FUNCTION_BLOCK FieldSignals (* CAT Function Block Type *)
  (* Standard: 61499-2 *)
  (* Version 0.0, 3/5/2026, Schneider Electric, template *)
  PACKAGE SE.Nereda;
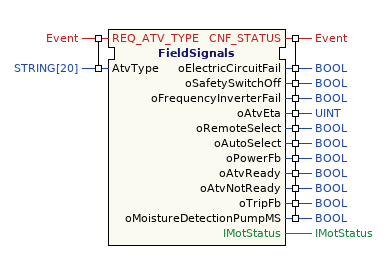
  EVENT_INPUT
    REQ_ATV_TYPE WITH AtvType;
  END_EVENT
  EVENT_OUTPUT
    CNF_STATUS WITH oElectricCircuitFail, oSafetySwitchOff, oFrequencyInverterFail, oAtvEta, oRemoteSelect, oAutoSelect, oPowerFb, oAtvReady, oAtvNotReady, oTripFb, oMoistureDetectionPumpMS;
  END_EVENT
  VAR_INPUT
    AtvType : STRING[20];
  END_VAR
  VAR_OUTPUT
    oElectricCircuitFail : BOOL; (* Current value(i) in the named variable array element *)
    oSafetySwitchOff : BOOL; (* Current value(i) in the named variable array element *)
    oFrequencyInverterFail : BOOL; (* Current value(i) in the named variable array element *)
    oAtvEta : UINT; (* Current value(i) in the named variable array element *)
    oRemoteSelect : BOOL; (* Current value(i) in the named variable array element *)
    oAutoSelect : BOOL; (* Current value(i) in the named variable array element *)
    oPowerFb : BOOL; (* Current value(i) in the named variable array element *)
    oAtvReady : BOOL; (* Current value(i) in the named variable array element *)
    oAtvNotReady : BOOL; (* Current value(i) in the named variable array element *)
    oTripFb : BOOL; (* Current value(i) in the named variable array element *)
    oMoistureDetectionPumpMS : BOOL;
  END_VAR
  PLUGS
    IMotStatus : IMotStatus;
  END_PLUGS
  (* 03 - FIELD INTERFACE IN *)
  (* 02 - FUNCTIONNAL OUTPUT INTERFACE *)
  (* 00 - INITIALIZATION *)
  (* 05 - LOGIC *)
  (* 04 - FIELD INTERFACE OUT *)
  (* 06 - HMI INTERFACE *)
  (* 01 - FUNCTIONNAL INPUT INTERFACE *)
  FBS
    INIT : plcStart(Prio := 24, Delay := T#0ms);
    ElectricCircuitFail : SYMLINKMULTIVARDST_1559B0FF8170C9BA0(QI := TRUE, NAME1 := '$${PATH}ElectricCircuitFail'); {SET_ATTRIBUTE(Configuration.GenericFBType.InterfaceParams, Runtime.System#I:=1;VALUE${I$}:BOOL)}
    SafetySwitchOff : SYMLINKMULTIVARDST_1559B0FF8170C9BA0(QI := TRUE, NAME1 := '$${PATH}SafetySwitchOff'); {SET_ATTRIBUTE(Configuration.GenericFBType.InterfaceParams, Runtime.System#I:=1;VALUE${I$}:BOOL)}
    FrequencyInverterFail : SYMLINKMULTIVARDST_1559B0FF8170C9BA0(QI := TRUE, NAME1 := '$${PATH}FrequencyInverterFail'); {SET_ATTRIBUTE(Configuration.GenericFBType.InterfaceParams, Runtime.System#I:=1;VALUE${I$}:BOOL)}
    ResetError_ATV3 : AtvResetError;
    ATV_ETA : SYMLINKMULTIVARDST_97F4072E4C409BE(QI := TRUE, NAME1 := '$${PATH}ATV_ETA'); {SET_ATTRIBUTE(Configuration.GenericFBType.InterfaceParams, Runtime.System#I:=1;VALUE${I$}:UINT)}
    ATV_Command : SYMLINKMULTIVARSRC_277E97BEC1451D2C(QI := TRUE, NAME1 := '$${PATH}ResetError_ATV', NAME2 := '$${PATH}CmdReady'); {SET_ATTRIBUTE(Configuration.GenericFBType.InterfaceParams, Runtime.System#I:=2;VALUE${I$}:BOOL,BOOL)}
    IThis : FieldSignals_HMI(QI := TRUE);
    RemoteSelect : SYMLINKMULTIVARDST_1559B0FF8170C9BA0(QI := TRUE, NAME1 := '$${PATH}RemoteSelect'); {SET_ATTRIBUTE(Configuration.GenericFBType.InterfaceParams, Runtime.System#I:=1;VALUE${I$}:BOOL)}
    AutoSelect : SYMLINKMULTIVARDST_1559B0FF8170C9BA0(QI := TRUE, NAME1 := '$${PATH}AutoSelect'); {SET_ATTRIBUTE(Configuration.GenericFBType.InterfaceParams, Runtime.System#I:=1;VALUE${I$}:BOOL)}
    PowerFb : SYMLINKMULTIVARDST_1559B0FF8170C9BA0(QI := TRUE, NAME1 := '$${PATH}PowerFb'); {SET_ATTRIBUTE(Configuration.GenericFBType.InterfaceParams, Runtime.System#I:=1;VALUE${I$}:BOOL)}
    AtvReady : SYMLINKMULTIVARDST_1559B0FF8170C9BA0(QI := TRUE, NAME1 := '$${PATH}AtvReady'); {SET_ATTRIBUTE(Configuration.GenericFBType.InterfaceParams, Runtime.System#I:=1;VALUE${I$}:BOOL)}
    EO_STATUS : E_MERGE_12;
    AtvNotReady : NOT_42C76073DCEB1A7A; {SET_ATTRIBUTE(Configuration.GenericFBType.InterfaceParams, Runtime.Standard#CNT:=1;OUT${CNT$}:BOOL)}
    RemoteAutoSelectMng : RemoteAutoMng;
    SelElectricCircuitFail : SELECT_81F91C08E00C8B28; {SET_ATTRIBUTE(Configuration.GenericFBType.InterfaceParams, Runtime.Standard#CNT:=2;SELECT:BOOL;IN${CNT$}:BOOL)}
    SelSafetySwitchOff : SELECT_81F91C08E00C8B28; {SET_ATTRIBUTE(Configuration.GenericFBType.InterfaceParams, Runtime.Standard#CNT:=2;SELECT:BOOL;IN${CNT$}:BOOL)}
    SelFrequencyInverterFail : SELECT_81F91C08E00C8B28; {SET_ATTRIBUTE(Configuration.GenericFBType.InterfaceParams, Runtime.Standard#CNT:=2;SELECT:BOOL;IN${CNT$}:BOOL)}
    SelATV_ETA : SELECT_32E1B08D4B0D0FE1; {SET_ATTRIBUTE(Configuration.GenericFBType.InterfaceParams, Runtime.Standard#CNT:=2;SELECT:BOOL;IN${CNT$}:UINT)}
    SelRemoteSelect : SELECT_81F91C08E00C8B28; {SET_ATTRIBUTE(Configuration.GenericFBType.InterfaceParams, Runtime.Standard#CNT:=2;SELECT:BOOL;IN${CNT$}:BOOL)}
    SelAutoSelect : SELECT_81F91C08E00C8B28; {SET_ATTRIBUTE(Configuration.GenericFBType.InterfaceParams, Runtime.Standard#CNT:=2;SELECT:BOOL;IN${CNT$}:BOOL)}
    SelPowerFb : SELECT_81F91C08E00C8B28; {SET_ATTRIBUTE(Configuration.GenericFBType.InterfaceParams, Runtime.Standard#CNT:=2;SELECT:BOOL;IN${CNT$}:BOOL)}
    SelAtvReady : SELECT_81F91C08E00C8B28; {SET_ATTRIBUTE(Configuration.GenericFBType.InterfaceParams, Runtime.Standard#CNT:=2;SELECT:BOOL;IN${CNT$}:BOOL)}
    NameGenerator : VALFORMAT_8708B18B173C5ABA(FORMAT := '%s', VALUE1 := '$${PATH:3,0}'); {SET_ATTRIBUTE(Configuration.GenericFBType.InterfaceParams, Runtime.Standard#I:=1;VALUE${I$}:STRING)}
    Frequency : SYMLINKMULTIVARDST_197068ABA215D7EBA(QI := TRUE, NAME1 := '$${PATH}MotorFrequecy'); {SET_ATTRIBUTE(Configuration.GenericFBType.InterfaceParams, Runtime.System#I:=1;VALUE${I$}:REAL)}
    PowerPercent_Sym : SYMLINKMULTIVARDST_197068ABA215D7EBA(QI := TRUE, NAME1 := '$${PATH}PowerPercent'); {SET_ATTRIBUTE(Configuration.GenericFBType.InterfaceParams, Runtime.System#I:=1;VALUE${I$}:REAL)}
    PowerCalculator : AtvPowerCalculator;
    TRIP : SYMLINKMULTIVARDST_1559B0FF8170C9BA0(QI := TRUE, NAME1 := '$${PATH}TRIP'); {SET_ATTRIBUTE(Configuration.GenericFBType.InterfaceParams, Runtime.System#I:=1;VALUE${I$}:BOOL)}
    SelTrip : SELECT_81F91C08E00C8B28; {SET_ATTRIBUTE(Configuration.GenericFBType.InterfaceParams, Runtime.Standard#CNT:=2;SELECT:BOOL;IN${CNT$}:BOOL)}
    MoistureDetectionPumpMS : SYMLINKMULTIVARDST_1559B0FF8170C9BA0(QI := TRUE, NAME1 := '$${PATH}MoistureDetectionPumpMS'); {SET_ATTRIBUTE(Configuration.GenericFBType.InterfaceParams, Runtime.System#I:=1;VALUE${I$}:BOOL)}
    SelMDPMS : SELECT_81F91C08E00C8B28; {SET_ATTRIBUTE(Configuration.GenericFBType.InterfaceParams, Runtime.Standard#CNT:=2;SELECT:BOOL;IN${CNT$}:BOOL)}
    NotElectricCircuitFail : NOT_42C76073DCEB1A7A; {SET_ATTRIBUTE(Configuration.GenericFBType.InterfaceParams, Runtime.Standard#CNT:=1;OUT${CNT$}:BOOL)}
    NOT1 : NOT_42C76073DCEB1A7A; {SET_ATTRIBUTE(Configuration.GenericFBType.InterfaceParams, Runtime.Standard#CNT:=1;OUT${CNT$}:BOOL)}
  END_FBS
  EVENT_CONNECTIONS
    ElectricCircuitFail.INITO TO SafetySwitchOff.INIT;
    SafetySwitchOff.INITO TO FrequencyInverterFail.INIT;
    FrequencyInverterFail.INITO TO ATV_ETA.INIT;
    ATV_ETA.INITO TO RemoteSelect.INIT;
    RemoteSelect.INITO TO AutoSelect.INIT;
    AutoSelect.INITO TO PowerFb.INIT;
    PowerFb.INITO TO AtvReady.INIT;
    SelAtvReady.CNF TO AtvNotReady.REQ;
    ElectricCircuitFail.CNF TO SelElectricCircuitFail.REQ;
    SafetySwitchOff.CNF TO SelSafetySwitchOff.REQ;
    FrequencyInverterFail.CNF TO SelFrequencyInverterFail.REQ;
    ATV_ETA.CNF TO SelATV_ETA.REQ;
    RemoteSelect.CNF TO SelRemoteSelect.REQ;
    AutoSelect.CNF TO SelAutoSelect.REQ;
    PowerFb.CNF TO SelPowerFb.REQ;
    AtvReady.CNF TO SelAtvReady.REQ;
    Frequency.INITO TO PowerPercent_Sym.INIT;
    AtvReady.INITO TO Frequency.INIT;
    PowerPercent_Sym.INITO TO TRIP.INIT;
    MoistureDetectionPumpMS.INITO TO ATV_Command.INIT;
    TRIP.CNF TO SelTrip.REQ;
    TRIP.INITO TO MoistureDetectionPumpMS.INIT;
    NOT1.CNF TO SelMDPMS.REQ;
    NotElectricCircuitFail.CNF TO IMotStatus.DA4A5AB166737E2B;
    SelSafetySwitchOff.CNF TO IMotStatus.SAF_SWT;
    SelFrequencyInverterFail.CNF TO IMotStatus.FREQ_FAIL;
    SelAtvReady.CNF TO IMotStatus.ATV_STE;
    SelRemoteSelect.CNF TO IMotStatus.REM_SEL;
    SelAutoSelect.CNF TO IMotStatus.AUTO_SEL;
    SelPowerFb.CNF TO IMotStatus.PWR_FB;
    SelTrip.CNF TO IMotStatus.8F309C1427B3D8B8;
    SelMDPMS.CNF TO IMotStatus.58CE25A170A20217;
    EO_STATUS.EO TO CNF_STATUS;
    NotElectricCircuitFail.CNF TO EO_STATUS.EI1;
    SelSafetySwitchOff.CNF TO EO_STATUS.EI2;
    SelFrequencyInverterFail.CNF TO EO_STATUS.EI3;
    SelATV_ETA.CNF TO EO_STATUS.EI4;
    RemoteAutoSelectMng.6BEF700BD5F898F8 TO EO_STATUS.EI5;
    SelPowerFb.CNF TO EO_STATUS.EI6;
    AtvNotReady.CNF TO EO_STATUS.523A3C57C3E4FA0F;
    SelTrip.CNF TO EO_STATUS.61E483B0D1B23F8E;
    SelMDPMS.CNF TO EO_STATUS.5434FC65F5B992C5;
    SelRemoteSelect.CNF TO RemoteAutoSelectMng.64070B2561E430BA;
    SelAutoSelect.CNF TO RemoteAutoSelectMng.64070B2561E430BA;
    PowerPercent_Sym.CNF TO PowerCalculator.REQ_POWER_PERC;
    REQ_ATV_TYPE TO PowerCalculator.REQ_ATV_TYPE;
    ATV_Command.INITO TO ResetError_ATV3.INIT;
    SelATV_ETA.CNF TO ResetError_ATV3.867B421BA90E2810;
    ResetError_ATV3.INITO TO INIT.ACK_FIRST;
    ResetError_ATV3.INITO TO NameGenerator.REQ;
    ResetError_ATV3.AD4F06CAB1B76C3D TO ATV_Command.REQ;
    ResetError_ATV3.3BE1C5BD951DD8A7 TO ATV_Command.REQ;
    SelElectricCircuitFail.CNF TO NotElectricCircuitFail.REQ;
    INIT.FIRST_INIT TO IThis.AD2A2FBE3D868A1D;
    INIT.REDO_INIT TO IThis.AD2A2FBE3D868A1D;
    PowerCalculator.CNF_POWER TO IThis.63337A003134C8E1;
    EO_STATUS.EO TO IThis.63337A003134C8E1;
    Frequency.CNF TO IThis.63337A003134C8E1;
    NameGenerator.CNF TO IThis.DAE3B0FAEAC06339;
    ResetError_ATV3.INITO TO IThis.213B97BD352AC6B9;
    IThis.047CDA631ACD0253 TO ElectricCircuitFail.INIT;
    IThis.9F0BB3507B1E4504 TO SelElectricCircuitFail.REQ;
    IThis.BE640CA1368FDF36 TO SelSafetySwitchOff.REQ;
    IThis.F7F6E0FF8EFA4B9E TO SelFrequencyInverterFail.REQ;
    IThis.1FE9183DAACAEFB7 TO SelATV_ETA.REQ;
    IThis.9B6E94ED39D931DA TO SelRemoteSelect.REQ;
    IThis.748EF2C5409B754A TO SelAutoSelect.REQ;
    IThis.DD989F023E0D2E7F TO SelPowerFb.REQ;
    IThis.C26243D045851266 TO SelAtvReady.REQ;
    IThis.DF011DEE9B6BC98A TO SelTrip.REQ;
    IThis.72F15890245A8D67 TO SelMDPMS.REQ;
    IThis.20926393FE3C273B TO SelElectricCircuitFail.REQ;
    IThis.20926393FE3C273B TO SelSafetySwitchOff.REQ;
    IThis.20926393FE3C273B TO SelFrequencyInverterFail.REQ;
    IThis.20926393FE3C273B TO SelATV_ETA.REQ;
    IThis.20926393FE3C273B TO SelRemoteSelect.REQ;
    IThis.20926393FE3C273B TO SelAutoSelect.REQ;
    IThis.20926393FE3C273B TO SelPowerFb.REQ;
    IThis.20926393FE3C273B TO SelAtvReady.REQ;
    IThis.20926393FE3C273B TO SelTrip.REQ;
    IThis.20926393FE3C273B TO SelMDPMS.REQ;
    AtvReady.CNF TO ResetError_ATV3.9E72FB83DA008EE6;
    MoistureDetectionPumpMS.CNF TO NOT1.REQ;
  END_CONNECTIONS
  DATA_CONNECTIONS
    NotElectricCircuitFail.OUT1 TO oElectricCircuitFail;
    SelSafetySwitchOff.OUT TO oSafetySwitchOff;
    SelFrequencyInverterFail.OUT TO oFrequencyInverterFail;
    SelATV_ETA.OUT TO oAtvEta;
    SelPowerFb.OUT TO oPowerFb;
    SelAtvReady.OUT TO oAtvReady;
    AtvNotReady.OUT1 TO oAtvNotReady;
    SelAtvReady.OUT TO AtvNotReady.IN1;
    ElectricCircuitFail.VALUE1 TO SelElectricCircuitFail.IN1;
    SafetySwitchOff.VALUE1 TO SelSafetySwitchOff.IN1;
    FrequencyInverterFail.VALUE1 TO SelFrequencyInverterFail.IN1;
    ATV_ETA.VALUE1 TO SelATV_ETA.IN1;
    RemoteSelect.VALUE1 TO SelRemoteSelect.IN1;
    AutoSelect.VALUE1 TO SelAutoSelect.IN1;
    PowerFb.VALUE1 TO SelPowerFb.IN1;
    AtvReady.VALUE1 TO SelAtvReady.IN1;
    TRIP.VALUE1 TO SelTrip.IN1;
    SelTrip.OUT TO oTripFb;
    NOT1.OUT1 TO SelMDPMS.IN1;
    SelMDPMS.OUT TO oMoistureDetectionPumpMS;
    NotElectricCircuitFail.OUT1 TO IMotStatus.9BFF267744CD9FD6;
    SelSafetySwitchOff.OUT TO IMotStatus.78CB3852B3811624;
    SelFrequencyInverterFail.OUT TO IMotStatus.D764D50DE95B92F7;
    SelAtvReady.OUT TO IMotStatus.469BA920D864796D;
    RemoteAutoSelectMng.35EEAE8FF93B7DBA TO IMotStatus.EF0659DE8FA343F8;
    RemoteAutoSelectMng.A72D9DB047E13611 TO IMotStatus.1313714BCA2AD84D;
    SelPowerFb.OUT TO IMotStatus.DFE83B4BA65B6F23;
    SelTrip.OUT TO IMotStatus.56D1AD5F30D2DBE7;
    SelMDPMS.OUT TO IMotStatus.6ADAD9BF6A0BA01D;
    RemoteAutoSelectMng.35EEAE8FF93B7DBA TO oRemoteSelect;
    RemoteAutoSelectMng.A72D9DB047E13611 TO oAutoSelect;
    SelRemoteSelect.OUT TO RemoteAutoSelectMng.B7B4969BA24515DC;
    SelAutoSelect.OUT TO RemoteAutoSelectMng.F1A2D6FBF53580DC;
    PowerPercent_Sym.VALUE1 TO PowerCalculator.PowerPercent;
    AtvType TO PowerCalculator.5CC1D4617F64C731;
    SelATV_ETA.OUT TO ResetError_ATV3.1FA1D80F2131516F;
    ResetError_ATV3.532FFE820545899D TO ATV_Command.VALUE1;
    ResetError_ATV3.AAB4EED808C21F76 TO ATV_Command.VALUE2;
    SelElectricCircuitFail.OUT TO NotElectricCircuitFail.IN1;
    NotElectricCircuitFail.OUT1 TO IThis.59E1B12ADD12039D;
    SelSafetySwitchOff.OUT TO IThis.78D88D59AF99C71A;
    SelFrequencyInverterFail.OUT TO IThis.E95314D83F614220;
    SelATV_ETA.OUT TO IThis.5E1721B0EFCCDD7A;
    SelRemoteSelect.OUT TO IThis.E774208D5A19204C;
    SelAutoSelect.OUT TO IThis.B58D6B2800878ECE;
    SelPowerFb.OUT TO IThis.8D45C0B812218232;
    SelAtvReady.OUT TO IThis.924CCF49C7E501AB;
    Frequency.VALUE1 TO IThis.F85EB7A00FC83BE7;
    PowerCalculator.PowerKW TO IThis.C9B2A692966C7391;
    NameGenerator.RESULT TO IThis.0179FB82468AB195;
    IThis.6F7AAC3E072B61BF TO SelElectricCircuitFail.SELECT;
    IThis.A333EA98BFBE0672 TO SelElectricCircuitFail.IN2;
    IThis.2ED6AD63DD1C0A2F TO SelSafetySwitchOff.SELECT;
    IThis.35685C36AB499CB1 TO SelSafetySwitchOff.IN2;
    IThis.7D1DBF3F0338AA78 TO SelFrequencyInverterFail.SELECT;
    IThis.CC6302DCC04BA25A TO SelFrequencyInverterFail.IN2;
    IThis.F6AE73A289A6D5CC TO SelATV_ETA.SELECT;
    IThis.FE5EA1F792072D33 TO SelATV_ETA.IN2;
    IThis.9A9E0B6AF830E4C9 TO SelRemoteSelect.SELECT;
    IThis.E0760EDFE472BD9D TO SelRemoteSelect.IN2;
    IThis.3F49DB4BAB98257E TO SelAutoSelect.SELECT;
    IThis.5810120BBF7661BD TO SelAutoSelect.IN2;
    IThis.36610EB6CE4B22E3 TO SelPowerFb.SELECT;
    IThis.0F40D5E3F72C391C TO SelPowerFb.IN2;
    IThis.05D63CC223B22EE0 TO SelAtvReady.SELECT;
    IThis.025681A258F0B88F TO SelAtvReady.IN2;
    IThis.D82D51A84BFAF967 TO SelTrip.SELECT;
    IThis.1D1919ADC2F64ABD TO SelTrip.IN2;
    IThis.169F5C2F236B0F72 TO SelMDPMS.SELECT;
    IThis.4DDD7D65F831BCFD TO SelMDPMS.IN2;
    AtvReady.VALUE1 TO ResetError_ATV3.9E07C1A3F72CEAED;
    MoistureDetectionPumpMS.VALUE1 TO NOT1.IN1;
  END_CONNECTIONS
END_FUNCTION_BLOCK
